{attribute addProperty BoxType "EP2316-0008-0016"}
{attribute addProperty Id "Set_safe_stateAT %Q*BOOL811Reset_outputsAT %Q*BOOL812"}
{attribute addProperty CRC "1934623490"}
{attribute addProperty SizeInBites "16"}
{attribute addProperty SizeInBytes "2"}
TYPE DO_Outputs_Device_73500302 :
STRUCT
	{attribute addProperty Name "Set_safe_state"}
	Set_safe_state AT %Q* : BOOL;
	{attribute addProperty Name "Reset_outputs"}
	Reset_outputs AT %Q* : BOOL;
END_STRUCT
END_TYPE

(* stored: Version 1.2.0.0, ProductVersion 3.1.4024.9
   DUT DO_Outputs_Device_73500302: Id {5ba700d4-99d8-4a81-9563-210112906e38} *)
